		internalEnable			:= FALSE;		
		IF internalDisable THEN
			internalDisable		:= FALSE;
			internalState		:= MV_BEGIN_HALTING;
			
		// Reset all commands issued by method calls
		ELSIF fbMoveAbsCA[0].Busy OR fbMoveAbsCA[0].CommandAborted THEN // OR fbMoveAbs.CommandAborted THEN
			fbMoveAbsCA[0].Execute		:= FALSE;
		ELSIF fbMoveAbsCA[1].Busy OR fbMoveAbsCA[1].CommandAborted THEN
			fbMoveAbsCA[1].Execute		:= FALSE;			
		ELSIF fbAddToGroup.Done THEN
			fbAddToGroup.Execute		:= FALSE;
		ELSIF fbMoveRelCA[0].Busy OR fbMoveRelCA[0].CommandAborted THEN
			fbMoveRelCA[0].Execute		:= FALSE;
		ELSIF fbMoveRelCA[1].Busy OR fbMoveRelCA[1].CommandAborted THEN
			fbMoveRelCA[1].Execute		:= FALSE;
		ELSIF fbGearInPosMoverCA[0].Busy OR fbGearInPosMoverCA[0].CommandAborted THEN
			fbGearInPosMoverCA[0].Execute	:= FALSE;
		ELSIF fbGearInPosMoverCA[1].Busy OR fbGearInPosMoverCA[1].CommandAborted THEN
			fbGearInPosMoverCA[1].Execute	:= FALSE;
		ELSIF fbGearInPosAxisCA[0].Busy OR fbGearInPosAxisCA[0].CommandAborted THEN
			fbGearInPosAxisCA[0].Execute	:= FALSE;
		ELSIF fbGearInPosAxisCA[1].Busy OR fbGearInPosAxisCA[1].CommandAborted THEN
			fbGearInPosAxisCA[1].Execute	:= FALSE;
		ELSIF fbHaltCA.Busy OR fbHaltCA.CommandAborted OR fbHaltCA.Done THEN
			fbHaltCA.Execute			:= FALSE;
		// This is different than the other similar cases, since a Stop command should prevent other commands from overriding it, thus
		// the Execute needs to remain High until the command has fully completed.
		ELSIF fbGroupStop.Done THEN
			fbGroupStop.Execute			:= FALSE;
		END_IF;
		
		THIS^.CyclicTrack();
		
		IF (internalReissue) THEN
			THIS^.SourceInstancePath	:= 'ReissueCommand';

			CASE internalCurrentMoveType OF
				MOVETYPE_NONE:
					// No current command to reissue	
				MOVETYPE_POSITION:
					THIS^.MoveToPosition( internalCurrentDestPosition );
				MOVETYPE_STATION:
					THIS^.MoveToStation( internalCurrentDestStation );
				MOVETYPE_VELOCITY:
					THIS^.MoveVelocity( MotionParameters.Velocity );
				MOVETYPE_SYNC_MOVER:
					THIS^.SyncToMover( internalMasterMover, internalGap );
				MOVETYPE_SYNC_AXIS:
					// This command should perhaps not be compatible with Reissue command
			END_CASE
			internalReissue := FALSE;
		END_IF

		// And catch all internal function block errors
		IF fbMoveAbsCA[0].Error THEN
			ErrorID					:= fbMoveAbsCA[0].ErrorID;
			ErrorOrigin				:= CONCAT( InstancePath, '.fbMoveAbs[0]' );
			internalState			:= MV_ERROR;
		ELSIF fbMoveAbsCA[1].Error THEN
			ErrorID					:= fbMoveAbsCA[1].ErrorId;
			ErrorOrigin				:= CONCAT( InstancePath, '.fbMoveAbs[1]' );
			internalState			:= MV_ERROR;
		ELSIF fbAddToGroup.Error THEN
			ErrorID					:= fbAddToGroup.ErrorID;
			ErrorOrigin				:= CONCAT( InstancePath, '.fbAddToGroup' );
			internalState			:= MV_ERROR;
		ELSIF fbGroupStop.Error THEN
			ErrorID					:= fbGroupStop.ErrorId;
			ErrorOrigin				:= CONCAT( InstancePath, '.fbGroupStop' );
			internalState			:= MV_ERROR;
		ELSIF fbMoveRelCA[0].Error THEN
			ErrorID					:= fbMoveRelCA[0].ErrorID;
			ErrorOrigin 			:= CONCAT ( InstancePath, '.fbMoveRelCA[0]');
			internalState			:= MV_ERROR;
		ELSIF fbMoveRelCA[1].Error THEN
			ErrorID					:= fbMoveRelCA[1].ErrorID;
			ErrorOrigin 			:= CONCAT ( InstancePath, '.fbMoveRelCA[1]');
			internalState			:= MV_ERROR;
		ELSIF fbReadStatus.Valid AND fbReadStatus.ErrorStop THEN
			ErrorID					:= fbReadStatus.Status.ErrorID;
			ErrorOrigin				:= CONCAT( InstancePath, '.fbReadStatus' );
			internalState			:= MV_ERROR;
		ELSIF fbGearInPosMoverCA[0].Error THEN
			ErrorID					:= fbGearInPosMoverCA[0].ErrorId;
			ErrorOrigin				:= CONCAT( InstancePath, '.fbGearInPosMoverCA[0]');
			internalState			:= MV_ERROR;
		ELSIF fbGearInPosMoverCA[1].Error THEN
			ErrorID					:= fbGearInPosMoverCA[1].ErrorId;
			ErrorOrigin				:= CONCAT( InstancePath, '.fbGearInPosMoverCA[1]');
			internalState			:= MV_ERROR;
		ELSIF fbGearInPosAxisCA[0].Error THEN
			ErrorID					:= fbGearInPosAxisCA[0].ErrorId;
			ErrorOrigin				:= CONCAT( InstancePath, '.fbGearInPosAxisCA[0]');
			internalState			:= MV_ERROR;
		ELSIF fbGearInPosAxisCA[1].Error THEN
			ErrorID					:= fbGearInPosAxisCA[1].ErrorId;
			ErrorOrigin				:= CONCAT( InstancePath, '.fbGearInPosAxisCA[1]');
			internalState			:= MV_ERROR;			
		ELSIF fbActivateTrack.Error THEN
			ErrorID					:= fbActivateTrack.ErrorId;
			ErrorOrigin				:= CONCAT( InstancePath, '.fbActivateTrack');
			internalState			:= MV_ERROR;
		END_IF
		
	MV_BEGIN_HALTING:	// --------------------------------------------------- begin stopping process
	
		Ready	:= FALSE;
		Busy	:= TRUE;
		Error	:= FALSE;
		ErrorID	:= 0;
		
		// Kill any active motion commands
		fbMoveRelCA[0].Execute		:= FALSE;
		fbMoveRelCA[1].Execute		:= FALSE;
		fbMoveAbsCA[0].Execute		:= FALSE;
		fbMoveAbsCA[1].Execute		:= FALSE;
				
		IF fbReadStatus.ErrorStop = FALSE THEN
			fbHaltCA.Execute		:= TRUE;
			//fbHaltCA.Deceleration	:= MotionParameters.Deceleration;
			//fbHaltCA.Jerk			:= MotionParameters.Jerk;
		ELSE
			internalState			:= MV_REMOVEFROMGROUP;
		END_IF;
		
		IF fbHaltCA.Active OR fbHaltCA.Done THEN
			internalState			:= MV_HALTING;
		ELSIF fbHaltCA.Error THEN
			ErrorID					:= fbHaltCA.ErrorID;
			ErrorOrigin				:= CONCAT( InstancePath, '.fbHalt' );
			internalState			:= MV_ERROR;				
		END_IF	
		
	MV_HALTING:	// ------------------------------------------------------- mover disabling
	
		Ready	:= FALSE;
		Busy	:= TRUE;
		Error	:= FALSE;
		ErrorID	:= 0;

		// Wait for the stopping action to complete
		IF fbHaltCA.Done THEN
			fbHaltCA.Execute		:= FALSE;
			internalState			:= MV_REMOVEFROMGROUP;
		ELSIF fbHaltCA.Error THEN
			ErrorID					:= fbStop.ErrorID;
			ErrorOrigin				:= CONCAT( InstancePath, '.fbHalt' );
			internalState			:= MV_ERROR;
		END_IF	
		
	MV_REMOVEFROMGROUP:	// ---------------------------------------------------- remove mover from CA group
	
		Ready	:= FALSE;
		Busy	:= TRUE;
		Error	:= FALSE;
		ErrorID	:= 0;
		
		fbRemoveFromGroup.Execute			:= TRUE;
		fbRemoveFromGroup.IdentInGroup		:= UDINT_TO_IDENTINGROUP( IdentInGroup );
		
		IF fbRemoveFromGroup.Done THEN
			fbRemoveFromGroup.Execute		:= FALSE;
			internalState					:= MV_DISABLING;
		END_IF
		


	MV_DISABLING:	// ----------------------------------------------------- start the disabling process

		Ready	:= FALSE;
		Busy	:= TRUE;
		Error	:= FALSE;
		ErrorID	:= 0;
		
		fbPower.Enable				:= FALSE;
		fbPower.Enable_Positive		:= FALSE;
		fbPower.Enable_Negative		:= FALSE;
		fbPower.BufferMode			:= MC_Aborting;
		fbPower.Override			:= 100;
			
		IF fbPower.Status = FALSE THEN
			internalState			:= MV_IDLE;
		ELSIF fbPower.Error THEN
			ErrorID					:= fbPower.ErrorID;
			ErrorOrigin				:= CONCAT( InstancePath, '.fbPower' );
			internalState			:= MV_ERROR;
		END_IF		
	
	MV_ERROR: // ------------------------------------------------------- mover in error state
	
		Ready	:= FALSE;
		Busy	:= FALSE;
		Error	:= TRUE;
		
		internalEnable			:= FALSE;		
		IF internalDisable THEN
			internalDisable		:= FALSE;
			internalState		:= MV_REMOVEFROMGROUP;
			ErrorOrigin			:= '';
		END_IF
		
END_CASE

fbPower( Axis := AxisReference );
fbReset( Axis := AxisReference );
fbStop( Axis := AxisReference );

fbHaltCA( Axis := AxisReference );
//fbDisable( Axis := AxisRef );
//fbExternEnable( Axis := AxisRef );

fbAddToGroup( AxesGroup := GroupReference, Axis := AxisReference );
fbRemoveFromGroup( AxesGroup := GroupReference );

fbGroupStatus( AxesGroup := GroupReference );
fbGroupEnable( AxesGroup := GroupReference );
fbGroupReset( AxesGroup := GroupReference );
fbGroupStop( AxesGroup := GroupReference );

fbMoveAbsCA[0]( Axis := AxisReference );
fbMoveAbsCA[1]( Axis := AxisReference );
fbReadStatus( Enable := TRUE, Axis := AxisReference );
fbMoveRelCA[0] ( Axis := AxisReference );
fbMoveRelCA[1] ( Axis := AxisReference );

fbGearInPosMoverCA[0]( Master := internalMasterMover.AxisReference, Slave := THIS^.AxisReference );
fbGearInPosMoverCA[1]( Master := internalMasterMover.AxisReference, Slave := THIS^.AxisReference );

fbGearInPosAxisCA[0]( Master := internalMasterAxis, Slave := THIS^.AxisReference );
fbGearInPosAxisCA[1]( Master := internalMasterAxis, Slave := THIS^.AxisReference );

fbReadM1DetectMode();
fbReadM1DetectValid();
fbReadM1DetectActive();
fbWriteM1Detect();

// track management
fbActivateTrack(Axis := AxisReference);
fbReadTrackPositions(Axis := AxisReference);
END_METHOD

METHOD CyclicTrack : BOOL
VAR
END_VAR
VAR_INST
	MsgCreate			: FB_TcMessage;	
END_VAR
// called by .Cyclic() to handle the MC_ActivateTrack call's required state machine
// this is only called while the mover is in the RUN state within .Cyclic() by design
// calling the track management functions on disabled or errored movers that are not
// assigned to a group just causes the track management functions to throw more errors

CASE internalTrackState OF
	// wait for command
	TrackState.WAIT_FOR_COMMAND:
		IF (internalActivateTrackFlag) THEN
			// unregister mover from current track (logical tracking)
			IF (internalTrack <> 0) THEN
				internalTrack^.UnregisterMover(THIS^);
			END_IF;

			// set flags
			internalTrack := ADR(ErrorTrack);
			internalTrackIsReady := FALSE;

			// advance state
			internalTrackState := TrackState.SETUP_FUNCTION;
		END_IF
		
	// setup and call the function
	TrackState.SETUP_FUNCTION:
		fbActivateTrack.TrackId := internalActivatingTrack^.OTCID;
		fbActivateTrack.Execute := TRUE;
		IF (fbActivateTrack.Busy) THEN
			fbActivateTrack.Execute := FALSE;
			internalTrackState := TrackState.MONITOR_RESPONSE;
		END_IF
	
	// monitor response	
	TrackState.MONITOR_RESPONSE:
		IF (fbActivateTrack.Error) THEN
			internalTrackState := TrackState.ERROR;
		ELSIF (fbActivateTrack.Done) THEN
			internalTrackState := TrackState.REQUIRED_DELAY;
		END_IF;
	
	// required delay
	// the FB has returned .Done but the change has not yet propigated to the NC
	TrackState.REQUIRED_DELAY:
		internalTrackStateDelay.IN := TRUE;
		IF (internalTrackStateDelay.Q) THEN
			internalTrackStateDelay.IN := FALSE;
			internalTrackState := TrackState.CLEAN_UP;
		END_IF;
	
	// clean up flags
	TrackState.CLEAN_UP:
		internalTrack := internalActivatingTrack;
		internalActivatingTrack := ADR(ErrorTrack);
		internalTrackIsReady := TRUE;
		MsgCreate.CreateEx( TC_EVENTS.XtsBaseEventClass.MoverActivateTrackComplete, 0);
		MsgCreate.ipArguments.Clear().AddString(THIS^.InstancePath).AddInt(THIS^.CurrentTrack^.Id);
		MsgCreate.Send(0);
		internalTrackState := TrackState.WAIT_END;
		
	TrackState.ERROR:
		// reset execute
		fbActivateTrack.Execute := FALSE;
		// GVL.ERROR_TRACK is intentionally left in place
		// internalTrackIsReady is left at false
		// error is recorded in Cyclic()
		internalTrackState := TrackState.WAIT_END;
		
	TrackState.WAIT_END: 
		// falling edge detection for internalActivateTrackFlag
		IF (NOT internalActivateTrackFlag) THEN
			// register mover
			internalTrack^.RegisterMover(THIS^);
			internalTrackState := TrackState.WAIT_FOR_COMMAND;	
		END_IF
		internalActivateTrackFlag := FALSE;

END_CASE

// read back track information
IF (internalTrackIsReady) THEN
	// track info should be stable, call the block
	fbReadTrackPositions.Enable := TRUE;
	// copy data when ready
	IF (fbReadTrackPositions.Valid) THEN
		TrackInfo.TrackPosition := fbReadTrackPositions.TrackPosition;
		TrackInfo.PartPosition := fbReadTrackPositions.PartPosition;
		TrackInfo.TrackId := fbReadTrackPositions.TrackId;
		TrackInfo.PartId := fbReadTrackPositions.PartId;
	END_IF
ELSE
	// don't call function block to allow it to reset
	fbReadTrackPositions.Enable := FALSE;
END_IF


// a delay is required after MC_ActivateTrack returns .Done
internalTrackStateDelay(PT := T#10MS);
END_METHOD

METHOD Disable : iMover
VAR_INPUT
END_VAR
VAR
END_VAR
VAR_INST
	MsgCreate	: FB_TcMessage;	
END_VAR

IF internalState = MV_RUN OR internalState = MV_ERROR THEN

	// Sets an internal flag to advance the state machine
	internalDisable		:= TRUE;
	
	MsgCreate.CreateEx( TC_EVENTS.XtsBaseEventClass.MoverDisable,0 );
	MsgCreate.ipArguments.Clear().AddString(THIS^.InstancePath).AddString(THIS^.SourceInstancePath);
	MsgCreate.Send(0);	
END_IF

THIS^.SourceInstancePath	:= 'Direct access';

Disable		:= THIS^;
END_METHOD

METHOD Enable : iMover
VAR_INPUT
END_VAR
VAR
END_VAR
VAR_INST
	MsgCreate	: FB_TcMessage;	
END_VAR

IF internalState = MV_IDLE THEN

	// Sets an internal flag to advance the state machine
	internalEnable		:= TRUE;
	
	MsgCreate.CreateEx( TC_EVENTS.XtsBaseEventClass.MoverEnable,0 );
	MsgCreate.ipArguments.Clear().AddString(THIS^.InstancePath).AddString(THIS^.SourceInstancePath);
	MsgCreate.Send(0);

END_IF;

THIS^.SourceInstancePath	:= 'Direct access';

Enable := THIS^;
END_METHOD

METHOD GroupStop : iMover
VAR_INPUT
END_VAR
VAR
	newCallTime	: LREAL;
END_VAR
VAR_INST
	MsgCreate	: FB_TcMessage;	
END_VAR


IF NOT( Ready ) THEN	// if the mover is not ready & able to accept a GroupHalt Command

	internalState	:= MV_ERROR;
	ErrorID			:= 19201;

ELSE	// otherwise execute the command
	
	// grab a timestamp of the command
	newCallTime		:= ULINT_TO_LREAL(F_GetSystemTime())/1E7;
	
	fbGroupStop.Execute			:= TRUE;
	fbGroupStop.Deceleration	:= MotionParameters.Deceleration;
	fbGroupStop.Jerk			:= MotionParameters.Jerk;
	
	memset( ADR( internalCurrentDestObjective ), 0, SIZEOF( internalCurrentDestObjective ));
	internalCurrentMoveType		:= MoverCommandType_enum.MOVETYPE_NONE;
	
END_IF

IF ( newCallTime - lastCallGroupStop ) > 1 THEN
	MsgCreate.CreateEx( TC_EVENTS.XtsBaseEventClass.MoverGroupStop,0 );
	MsgCreate.ipArguments.Clear().AddString(THIS^.InstancePath).AddString(THIS^.SourceInstancePath);
	MsgCreate.Send(0);
END_IF

THIS^.SourceInstancePath	:= 'Direct access';

lastCallGroupStop	:= newCallTime;

GroupStop		:= THIS^;
END_METHOD

METHOD Halt : iMover
VAR_INPUT
END_VAR
VAR
	newCallTime: LREAL;
END_VAR
VAR_INST
	MsgCreate: FB_TcMessage;	
END_VAR

IF NOT( Ready ) THEN
	
	internalState	:= MV_ERROR;
	ErrorID			:= 19201;
	
ELSIF fbHaltCA.Busy THEN	

	newCallTime		:= ULINT_TO_LREAL(F_GetSystemTime())/1E7;
	
	// oddly, MC_HaltCA does not include an option for BufferMode
	// so do nothing
	
ELSE
	
	newCallTime		:= ULINT_TO_LREAL(F_GetSystemTime())/1E7;
	
	fbHaltCA.Execute		:= TRUE;
	fbHaltCA.Deceleration	:= MotionParameters.Deceleration;
	fbHaltCA.Jerk			:= MotionParameters.Jerk;
	
	fbHaltCA( Axis := AxisReference );
	
END_IF

internalCurrentMoveType		:= MOVETYPE_NONE;
internalCurrentDestPosition	:= 1E300;

memset( ADR( internalCurrentDestObjective), 0, SIZEOF( internalCurrentDestObjective ));
internalCurrentDestStation	REF= 0;

IF ( newCallTime - lastCallHalt ) > 1 THEN
	MsgCreate.CreateEx( TC_EVENTS.XtsBaseEventClass.MoverHalt,0);
	MsgCreate.ipArguments.Clear().AddString(THIS^.InstancePath).AddString(THIS^.SourceInstancePath).AddLReal(MotionParameters.Deceleration);
	MsgCreate.Send(0);
END_IF

THIS^.SourceInstancePath	:= 'Direct access';

lastCallHalt		:= newCallTIme;

Halt	:= THIS^;
END_METHOD

{attribute 'monitoring' := 'call'}
PROPERTY IsSyncedToAxis : BOOL
GET


IsSyncedToAxis		:= fbGearInPosAxisCA[0].InSync OR fbGearInPosAxisCA[1].InSync;
END_GET
END_PROPERTY

{attribute 'monitoring' := 'call'}
PROPERTY IsSyncedToMover : BOOL
GET


IsSyncedToMover		:= fbGearInPosMoverCA[0].InSync OR fbGearInPosMoverCA[1].InSync;
END_GET
END_PROPERTY

PROPERTY IsTrackReady : BOOL
GET
IsTrackReady := internalTrackIsReady;
END_GET
END_PROPERTY

METHOD LogUserEvent : iMover
VAR_INPUT
	String1	: STRING;	// First content section of user-event message
	String2 : STRING;	// Second content section of user-event message
	String3 : STRING;	// Third content section of user-event message
END_VAR
VAR
END_VAR
VAR_INST
	MsgCreate: FB_TcMessage;	
END_VAR



MsgCreate.CreateEx( TC_EVENTS.XtsBaseEventClass.UserEvent, 0 );
MsgCreate.ipArguments.Clear().AddString(String1).AddString(String2).AddString(String3);
MsgCreate.Send(0);

LogUserEvent	:= THIS^;
END_METHOD

PROPERTY MasterMover : Reference To Mover
GET


IF THIS^.internalCurrentMoveType = MOVETYPE_SYNC_MOVER THEN
	MasterMover		REF= internalMasterMover;
ELSE
	MasterMover		REF= 0;
END_IF
END_GET
END_PROPERTY

METHOD PUBLIC MoveToPosition : iMover
VAR_INPUT
	DestinationPosition		: LREAL;	// position on track for a shuttle to move towards
END_VAR
VAR
	newCallTime		: LREAL;
END_VAR
VAR_INST
	MsgCreate		: FB_TcMessage;	
END_VAR

IF NOT( Ready ) THEN	// if the mover is not ready & able to accept a moveabs command...
	
	internalState	:= MV_ERROR;
	ErrorID			:= 19201;
	
ELSE	// otherwise let 'er rip
	
	newCallTime		:= ULINT_TO_LREAL(F_GetSystemTime())/1E7;
	internalReissue := FALSE;	// reissue no longer necessary
	
	IF fbMoveAbsCA[0].Busy = FALSE THEN
		
		fbMoveAbsCA[0].Jerk			:= MotionParameters.Jerk;
		fbMoveAbsCA[0].Acceleration	:= MotionParameters.Acceleration;
		fbMoveAbsCA[0].Deceleration	:= MotionParameters.Deceleration;
		fbMoveAbsCA[0].Velocity		:= MotionParameters.Velocity;
		fbMoveAbsCA[0].Direction	:= MotionParameters.Direction;
		fbMoveAbsCA[0].Options.DynamicsReferenceSystem := CurrentTrack^.OTCID;
		fbMoveAbsCA[0].Options.PositionReferenceSystem := CurrentTrack^.OTCID;
		
		fbMoveAbsCA[0].Position		:= DestinationPosition;
		
		fbMoveAbsCA[0].BufferMode	:= mcAborting;
		fbMoveAbsCA[0].Execute		:= TRUE;
		 
		fbMoveAbsCA[0].Execute		:= TRUE;		// execute this block, and...
		fbMoveAbsCA[1].Execute		:= FALSE;		// if necessary, interrupt this one
		
		fbMoveAbsCA[0]( Axis := AxisReference );
		
	ELSIF fbMoveAbsCA[1].Busy = FALSE THEN
		
		fbMoveAbsCA[1].Jerk			:= MotionParameters.Jerk;
		fbMoveAbsCA[1].Acceleration	:= MotionParameters.Acceleration;
		fbMoveAbsCA[1].Deceleration	:= MotionParameters.Deceleration;
		fbMoveAbsCA[1].Velocity		:= MotionParameters.Velocity;
		fbMoveAbsCA[1].Direction	:= MotionParameters.Direction;
		fbMoveAbsCA[1].Options.DynamicsReferenceSystem := CurrentTrack^.OTCID;
		fbMoveAbsCA[1].Options.PositionReferenceSystem := CurrentTrack^.OTCID;

		
		fbMoveAbsCA[1].Position		:= DestinationPosition;
		
		fbMoveAbsCA[1].BufferMode	:= mcAborting;
		fbMoveAbsCA[1].Execute		:= TRUE;
		
		fbMoveAbsCA[1].Execute		:= TRUE;		// execute this block, and...
		fbMoveAbsCA[0].Execute		:= FALSE;		// if necessary, interrupt this one
		
		fbMoveAbsCA[1]( Axis := AxisReference );
		 
	ELSE
		MsgCreate.CreateEx( TC_EVENTS.XtsBaseEventClass.MoverMoveToPositionOverload,0 );
		MsgCreate.ipArguments.Clear().AddString(THIS^.InstancePath).AddString(THIS^.SourceInstancePath).AddLReal(DestinationPosition);
		MsgCreate.Send(0);
	END_IF
	
END_IF

internalCurrentMoveType		:= MOVETYPE_POSITION;
internalCurrentDestPosition := DestinationPosition;

memset( ADR( internalCurrentDestObjective ), 0, SIZEOF( internalCurrentDestObjective ));
internalCurrentDestStation	REF= 0;

IF ( newCallTime - lastCallMovePos ) > 1 THEN
	MsgCreate.CreateEx( TC_EVENTS.XtsBaseEventClass.MoverMoveToPosition,0 );
	MsgCreate.ipArguments.Clear().AddString(THIS^.InstancePath).AddString(THIS^.SourceInstancePath).AddLReal(DestinationPosition);
	MsgCreate.Send(0);
END_IF;

THIS^.SourceInstancePath	:= 'Direct access';

lastCallMovePos		:= newCallTime;

MoveToPosition		:= THIS^;
END_METHOD

METHOD MoveToStation : iMover
VAR_INPUT
	DestinationStation	: REFERENCE TO Station;	
END_VAR
VAR
	newCallTime			: LREAL;
END_VAR
VAR_INST
	MsgCreate			: FB_TcMessage;	
END_VAR
IF NOT( Ready ) AND NOT(__ISVALIDREF( DestinationStation )) THEN	// if the mover is not ready & able to accept a moveabs command...
	
	internalState	:= MV_ERROR;
	ErrorID			:= 19201;
	
ELSE	// otherwise let 'er rip
	
	newCallTime		:= ULINT_TO_LREAL(F_GetSystemTime())/1E7;
	internalReissue := FALSE;	// reissue no longer necessary
	
	IF fbMoveAbsCA[0].Busy = FALSE THEN
		
		fbMoveAbsCA[0].Jerk			:= MotionParameters.Jerk;
		fbMoveAbsCA[0].Acceleration	:= MotionParameters.Acceleration;
		fbMoveAbsCA[0].Deceleration	:= MotionParameters.Deceleration;
		fbMoveAbsCA[0].Velocity		:= MotionParameters.Velocity;
		fbMoveAbsCA[0].Direction	:= MotionParameters.Direction;
		fbMoveAbsCA[0].Options.DynamicsReferenceSystem := CurrentTrack^.OTCID;
		fbMoveAbsCA[0].Options.PositionReferenceSystem := CurrentTrack^.OTCID;
		
		fbMoveAbsCA[0].Position		:= DestinationStation.internalPosition;
		
		fbMoveAbsCA[0].BufferMode	:= mcAborting;
		fbMoveAbsCA[0].Execute		:= TRUE;
		 
		fbMoveAbsCA[0].Execute		:= TRUE;		// execute this block, and...
		fbMoveAbsCA[1].Execute		:= FALSE;		// if necessary, interrupt this one
		
		fbMoveAbsCA[0]( Axis := AxisReference );
		
	ELSIF fbMoveAbsCA[1].Busy = FALSE THEN
		
		fbMoveAbsCA[1].Jerk			:= MotionParameters.Jerk;
		fbMoveAbsCA[1].Acceleration	:= MotionParameters.Acceleration;
		fbMoveAbsCA[1].Deceleration	:= MotionParameters.Deceleration;
		fbMoveAbsCA[1].Velocity		:= MotionParameters.Velocity;
		fbMoveAbsCA[1].Direction	:= MotionParameters.Direction;
		fbMoveAbsCA[1].Options.DynamicsReferenceSystem := CurrentTrack^.OTCID;
		fbMoveAbsCA[1].Options.PositionReferenceSystem := CurrentTrack^.OTCID;
		
		fbMoveAbsCA[1].Position		:= DestinationStation.internalPosition;
		
		fbMoveAbsCA[1].BufferMode	:= mcAborting;
		fbMoveAbsCA[1].Execute		:= TRUE;
		
		fbMoveAbsCA[1].Execute		:= TRUE;		// execute this block, and...
		fbMoveAbsCA[0].Execute		:= FALSE;		// if necessary, interrupt this one

		fbMoveAbsCA[1]( Axis := AxisReference );	

	ELSE
		MsgCreate.CreateEx( TC_EVENTS.XtsBaseEventClass.MoverMoveToStationOverload,0 );
		MsgCreate.ipArguments.Clear().AddString(THIS^.InstancePath).AddString(THIS^.SourceInstancePath).AddString(DestinationStation.InstancePath);
		MsgCreate.Send(0);
		
	END_IF
	
	// Set the current destination object to the instance path of the objective, or 0 if unassigned
	internalCurrentDestPosition		:= DestinationStation.Position;
	internalCurrentDestObjective	:= SEL( __ISVALIDREF( DestinationStation ), '', DestinationStation.InstancePath );
	internalCurrentDestStation		REF= DestinationStation;
	internalCurrentMoveType			:= MOVETYPE_STATION;
	
	// Register this mover with the station, so the station knows this mover is incoming
	DestinationStation.RegisterMover( THIS^ );
	
END_IF

IF ( newCallTime - lastCallMoveSta ) > 1 THEN
	MsgCreate.CreateEx( TC_EVENTS.XtsBaseEventClass.MoverMoveToStation,0 );
	MsgCreate.ipArguments.Clear().AddString(THIS^.InstancePath).AddString(THIS^.SourceInstancePath).AddString(DestinationStation.InstancePath);
	MsgCreate.Send(0);
END_IF

THIS^.SourceInstancePath	:= 'Direct access';

lastCallMoveSta		:= newCallTime;

MoveToStation		:= THIS^;
END_METHOD

METHOD MoveVelocity : iMover
VAR_INPUT
	DesiredVelocity : LREAL;		//The velocity to be commanded [mm/s]
END_VAR
VAR
	negativeCommand	: BOOL;
	newCallTime		: LREAL;
END_VAR
VAR_INST
	MsgCreate		: FB_TcMessage;	
END_VAR
IF NOT ( ready ) THEN
	
	internalState	:= MV_ERROR;
	ErrorID			:= 19201;
	
ELSE
	
	newCallTime		:= ULINT_TO_LREAL(F_GetSystemTime())/1E7;
	internalReissue := FALSE;	// reissue no longer necessary
	
	negativeCommand					:= SEL( DesiredVelocity < 0, FALSE, TRUE );
	MotionParameters.Velocity		:= ABS( DesiredVelocity );
	
	IF fbMoveRelCA[0].Busy = FALSE THEN
		
		fbMoveRelCA[0].Jerk			:= MotionParameters.Jerk;
		
		fbMoveRelCA[0].Acceleration	:= MotionParameters.Acceleration;
		fbMoveRelCA[0].Deceleration	:= MotionParameters.Deceleration;
		fbMoveRelCA[0].Velocity		:= MotionParameters.Velocity;
		
		fbMoveRelCA[0].Distance		:= SEL( negativeCommand, 1E100, -1E100 );
		
		      
		fbMoveRelCA[0].BufferMode	:= mcAborting;
		      
		fbMoveRelCA[0].Execute		:= TRUE;		// execute this block, and...
		fbMoveRelCA[1].Execute		:= FALSE;		// if necessary, interrupt this one
		
		fbMoveRelCA[0]( Axis := AxisReference );
		
	ELSIF fbMoveRelCA[1].Busy = FALSE THEN
		
		fbMoveRelCA[1].Jerk			:= MotionParameters.Jerk;
		
		fbMoveRelCA[1].Acceleration	:= MotionParameters.Acceleration;
		fbMoveRelCA[1].Deceleration	:= MotionParameters.Deceleration;
		fbMoveRelCA[1].Velocity		:= MotionParameters.Velocity;
		      
		fbMoveRelCA[1].Distance		:= SEL( negativeCommand, 1E100, -1E100 );
		      
		fbMoveRelCA[1].BufferMode	:= mcAborting;
		      
		fbMoveRelCA[1].Execute		:= TRUE;		// execute this block, and...
		fbMoveRelCA[0].Execute		:= FALSE;		// if necessary, interrupt this one

		fbMoveRelCA[1]( Axis := AxisReference );
	ELSE
		MsgCreate.CreateEx( TC_EVENTS.XtsBaseEventClass.MoverMoveVelocityOverload,0 );
		MsgCreate.ipArguments.Clear().AddString(THIS^.InstancePath).AddString(THIS^.SourceInstancePath).AddLReal(DesiredVelocity);
		MsgCreate.Send(0);
	END_IF

END_IF

fbMoveRelCA[0] ( Axis := AxisReference );
fbMoveRelCA[1] ( Axis := AxisReference );


internalCurrentMoveType		:= MOVETYPE_VELOCITY;
internalCurrentDestPosition := 1E300;

memset( ADR( internalCurrentDestObjective ), 0, SIZEOF( internalCurrentDestObjective ));
internalCurrentDestStation	REF= 0;

IF ( newCallTime - lastCallMoveVel ) > 1 THEN
	MsgCreate.CreateEx( TC_EVENTS.XtsBaseEventClass.MoverMoveVelocity,0 );
	MsgCreate.ipArguments.Clear().AddString(THIS^.InstancePath).AddString(THIS^.SourceInstancePath).AddLReal(DesiredVelocity);
	MsgCreate.Send(0);
END_IF;

THIS^.SourceInstancePath	:= 'Direct access';

lastCallMoveVel		:= newCallTime;

MoveVelocity		:= THIS^;
END_METHOD

PROPERTY Payload : Payload_TYP;
GET


Payload	:= internalPayload;
END_GET
SET


internalPayload	:= Payload;
END_SET
END_PROPERTY

METHOD ReissueCommand : iMover
VAR_INPUT
END_VAR

// set flag for use in .Cyclic()
internalReissue := TRUE;


ReissueCommand		:= THIS^;
END_METHOD

METHOD SetAcceleration : iMover
VAR_INPUT
	Acceleration	: LREAL;
END_VAR
VAR
	newCallTime		: LREAL;
END_VAR
VAR_INST
	MsgCreate		: FB_TcMessage;	
END_VAR

newCallTime		:= ULINT_TO_LREAL(F_GetSystemTime())/1E7;

MotionParameters.Acceleration		:= LIMIT( 0, Acceleration, 1E300 );	// upper limit is capped by the axis object parameters

THIS^.ReissueCommand();

IF ( newCallTime - lastCallSetAcc ) > 1 THEN
	MsgCreate.CreateEx( TC_EVENTS.XtsBaseEventClass.MoverSetAcceleration,0 );
	MsgCreate.ipArguments.Clear().AddString(THIS^.InstancePath).AddString(THIS^.SourceInstancePath).AddLReal(Acceleration);
	MsgCreate.Send(0);
END_IF;

THIS^.SourceInstancePath	:= 'Direct access';

lastCallSetAcc		:= newCallTime;

SetAcceleration		:= THIS^;
END_METHOD

METHOD SetDeceleration : iMover
VAR_INPUT
	Deceleration	: LREAL;
END_VAR
VAR
	newCallTime		: LREAL;
END_VAR
VAR_INST
	MsgCreate		: FB_TcMessage;	
END_VAR

newCallTime		:= ULINT_TO_LREAL(F_GetSystemTime())/1E7;

MotionParameters.Deceleration	:= LIMIT( 0, Deceleration, 1E300 ); // upper limit is capped by the axis parameters

THIS^.ReissueCommand();

IF ( newCallTime - lastCallSetDec ) > 1 THEN
	MsgCreate.CreateEx( TC_EVENTS.XtsBaseEventClass.MoverSetDeceleration,0 );
	MsgCreate.ipArguments.Clear().AddString(THIS^.InstancePath).AddString(THIS^.SourceInstancePath).AddLReal(Deceleration);
	MsgCreate.Send(0);
END_IF

THIS^.SourceInstancePath	:= 'Direct access';

lastCallSetDec		:= newCallTime;

SetDeceleration		:= THIS^;
END_METHOD

METHOD SetDirection : iMover
VAR_INPUT
	Direction		: Tc3_Mc3Definitions.MC_Direction;
END_VAR
VAR
	newCallTime		: LREAL;
END_VAR
VAR_INST
	MsgCreate		: FB_TcMessage;	
END_VAR

newCallTime		:= ULINT_TO_LREAL(F_GetSystemTime())/1E7;

MotionParameters.Direction		:= Direction;

THIS^.ReissueCommand();

IF ( newCallTime - lastCallSetDir ) > 1 THEN
	MsgCreate.CreateEx( TC_EVENTS.XtsBaseEventClass.MoverSetDirection,0 );
	MsgCreate.ipArguments.Clear().AddString(THIS^.InstancePath).AddString(THIS^.SourceInstancePath).AddInt(Direction);
	MsgCreate.Send(0);
END_IF

THIS^.SourceInstancePath	:= 'Direct access';

lastCallSetDir		:= newCallTime;

SetDirection		:= THIS^;
END_METHOD

METHOD SetJerk : iMover
VAR_INPUT
	Jerk		: LREAL;
END_VAR
VAR
	newCallTime	: LREAL;
END_VAR
VAR_INST
	MsgCreate	: FB_TcMessage;	
END_VAR

newCallTime		:= ULINT_TO_LREAL(F_GetSystemTime())/1E7;

MotionParameters.Jerk		:= LIMIT( 0, Jerk, 1E300 ); // upper limit is capped by the axis parameters

THIS^.ReissueCommand();

IF ( newCallTime - lastCallSetJerk ) > 1 THEN
	MsgCreate.CreateEx( TC_EVENTS.XtsBaseEventClass.MoverSetJerk,0 );
	MsgCreate.ipArguments.Clear().AddString(THIS^.InstancePath).AddString(THIS^.SourceInstancePath).AddLReal(Jerk);
	MsgCreate.Send(0);
END_IF

THIS^.SourceInstancePath	:= 'Direct access';

lastCallSetJerk		:= newCallTIme;

SetJerk		:= THIS^;
END_METHOD

METHOD SetVelocity : iMover
VAR_INPUT
	Velocity		: LREAL;		// Updates Mover's internal velocity parameter. Takes effect immediately. [mm/s]
END_VAR
VAR
	logstr			: STRING(200);		// method variable containing an event log message for the command
	LogEvent		: INT;
	newCallTime		: LREAL;
END_VAR
VAR_INST
	MsgCreate		: FB_TcMessage;	
END_VAR

newCallTime		:= ULINT_TO_LREAL(F_GetSystemTime())/1E7;

MotionParameters.Velocity	:= LIMIT( 0, Velocity, 1E300 ); // upper limit is capped by the axis parameters 

THIS^.ReissueCommand();

IF ( newCallTime - lastCallSetVel ) > 1 THEN
	MsgCreate.CreateEx( TC_EVENTS.XtsBaseEventClass.MoverSetVelocity,0 );
	MsgCreate.ipArguments.Clear().AddString(THIS^.InstancePath).AddString(THIS^.SourceInstancePath).AddLReal(Velocity);
	MsgCreate.Send(0);
END_IF

THIS^.SourceInstancePath	:= 'Direct access';

lastCallSetVel	:= newCallTime;

SetVelocity		:= THIS^;
END_METHOD

METHOD SyncToAxis : iMover
VAR_INPUT
	
	MasterAxis		: REFERENCE TO AXIS_REF;
	MasterSyncPos	: LREAL;				// Master sync position (nonmodulo), where the input axis will be located when first synchronized
	SlaveSyncPos	: LREAL;				// Mover sync position, where the mover will be located when first synchronized
	SyncStrategy	: MC_SYNC_STRATEGY;		// Direction input
	
END_VAR
VAR
	newCallTime		: LREAL;
END_VAR
VAR_INST
	MsgCreate		: FB_TcMessage;
END_VAR


IF NOT( Ready ) THEN
	
	internalState		:= MV_ERROR;
	ErrorID				:= 19201;
	
ELSE
	
	newCallTime			:= ULINT_TO_LREAL(F_GetSystemTime())/1E7;
	internalReissue := FALSE;	// reissue no longer necessary
	
	internalMasterAxis		REF= MasterAxis;
	
	IF fbGearInPosAxisCA[0].Busy = FALSE THEN
		
		fbGearInPosAxisCA[0].Execute			:= TRUE;
		
		fbGearInPosAxisCA[0].RatioNumerator		:= 1;
		fbGearInPosAxisCA[0].RatioDenumerator	:= 1;
		
		fbGearInPosAxisCA[0].MasterSyncPosition	:= MasterSyncPos;	// This needs to be nonmodulo
		fbGearInPosAxisCA[0].SlaveSyncPosition	:= SlaveSyncPos;
		
		fbGearInPosAxisCA[0].SyncStrategy		:= SyncStrategy;
		
		fbGearInPosAxisCA[0].Options.DynamicsReferenceSystem := CurrentTrack^.OTCID;
		fbGearInPosAxisCA[0].Options.SlaveSyncPositionReferenceSystem := CurrentTrack^.OTCID;

		
		IF MotionParameters.Direction = mcDirectionPositive THEN
			fbGearInPosAxisCA[0].SyncMode		:= mcSyncModePositive;
		ELSIF MotionParameters.Direction = mcDirectionNegative THEN
			fbGearInPosAxisCA[0].SyncMode		:= mcSyncModeNegative;
		END_IF
		
		fbGearInPosAxisCA[0].Velocity			:= MotionParameters.Velocity;
		fbGearInPosAxisCA[0].Acceleration		:= MotionParameters.Acceleration;
		fbGearInPosAxisCA[0].Deceleration		:= MotionParameters.Deceleration;
		fbGearInPosAxisCA[0].Jerk				:= MotionParameters.Jerk;
		
		fbGearInPosAxisCA[0].BufferMode			:= Tc3_Mc3Definitions.MC_BUFFER_MODE.mcAborting;
		
		fbGearInPosAxisCA[0]( Master := MasterAxis, Slave := THIS^.AxisReference );		
		
	ELSIF fbGearInPosAxisCA[1].Busy = FALSE THEN
		
		fbGearInPosAxisCA[1].Execute			:= TRUE;
		
		fbGearInPosAxisCA[1].RatioNumerator		:= 1;
		fbGearInPosAxisCA[1].RatioDenumerator	:= 1;
		
		fbGearInPosAxisCA[1].MasterSyncPosition	:= MasterSyncPos;	// This needs to be nonmodulo
		fbGearInPosAxisCA[1].SlaveSyncPosition	:= SlaveSyncPos;
		
		fbGearInPosAxisCA[1].SyncStrategy		:= SyncStrategy;
		
		fbGearInPosAxisCA[1].Options.DynamicsReferenceSystem := CurrentTrack^.OTCID;
		fbGearInPosAxisCA[1].Options.SlaveSyncPositionReferenceSystem := CurrentTrack^.OTCID;
		
		IF MotionParameters.Direction = mcDirectionPositive THEN
			fbGearInPosAxisCA[1].SyncMode		:= mcSyncModePositive;
		ELSIF MotionParameters.Direction = mcDirectionNegative THEN
			fbGearInPosAxisCA[1].SyncMode		:= mcSyncModeNegative;				
		END_IF
		
		fbGearInPosAxisCA[1].Velocity			:= MotionParameters.Velocity;
		fbGearInPosAxisCA[1].Acceleration		:= MotionParameters.Acceleration;
		fbGearInPosAxisCA[1].Deceleration		:= MotionParameters.Deceleration;
		fbGearInPosAxisCA[1].Jerk				:= MotionParameters.Jerk;
		
		fbGearInPosAxisCA[1].BufferMode			:= Tc3_Mc3Definitions.MC_BUFFER_MODE.mcAborting;
		
		fbGearInPosAxisCA[1]( Master := MasterAxis, Slave := THIS^.AxisReference );

	ELSE
		MsgCreate.CreateEx( TC_EVENTS.XtsBaseEventClass.MoverSyncToAxisOverload, 0 );
		MsgCreate.ipArguments.Clear().AddString(THIS^.InstancePath).AddString(THIS^.SourceInstancePath);
		MsgCreate.Send(0);
	END_IF
	
END_IF

internalCurrentMoveType			:= MOVETYPE_SYNC_AXIS;
internalCurrentDestPosition		:= 1E300;

memset( ADR( internalCurrentDestObjective ), 0, SIZEOF( internalCurrentDestObjective ));
internalCurrentDestStation		REF= 0;

IF ( newCallTime - lastCallSync ) > 1 THEN
	MsgCreate.CreateEx( TC_EVENTS.XtsBaseEventClass.MoverSyncToAxis, 0 );
	MsgCreate.ipArguments.Clear().AddString(THIS^.InstancePath).AddString(THIS^.SourceInstancePath);
	MsgCreate.Send(0);
END_IF

THIS^.SourceInstancePath		:= 'Direct access';

lastCallSync	:= newCallTime;

SyncToAxis		:= THIS^;
END_METHOD

METHOD SyncToMover : iMover
VAR_INPUT
	MasterMover			: REFERENCE TO Mover;	// Synchronization master mover, whose position to follow. Further motion commands break the pairing
	Gap					: LREAL;				// Gap distance to lead mover. Positive values indicate following, negative values indicate leading
END_VAR
VAR
	CWDistToSync		: LREAL;
	CWDistToMaster		: LREAL;
	syncPos				: LREAL;
	newCallTime			: LREAL;
END_VAR
VAR_INST
	MsgCreate			: FB_TcMessage;	
END_VAR
IF NOT( Ready ) THEN

	internalState	:= MV_ERROR;
	ErrorID			:= 19201;
	
ELSE	// let 'er rip
	
	newCallTime		:= ULINT_TO_LREAL(F_GetSystemTime())/1E7;
	internalReissue := FALSE;	// reissue no longer necessary

	internalMasterMover		REF= MasterMover;
	internalGap				:= Gap;
	
	
	syncPos			:= internalMasterMover.AxisReference.NcToPlc.ActPos - internalGap;
	CWDistToSync	:= MODABS( syncPos - THIS^.AxisReference.NcToPlc.ActPos, GVL.TRACK_LENGTH );
	CWDistToMaster	:= MODABS( internalMasterMover.AxisReference.NcToPlc.ActPos - THIS^.AxisReference.NcToPlc.ActPos, GVL.TRACK_LENGTH );
		
	IF fbGearInPosMoverCA[0].Busy = FALSE THEN
		
		fbGearInPosMoverCA[0].Execute				:= TRUE;
			
		fbGearInPosMoverCA[0].RatioNumerator			:= 1;
		fbGearInPosMoverCA[0].RatioDenumerator		:= 1;
		
		fbGearInPosMoverCA[0].MasterSyncPosition		:= internalMasterMover.AxisReference.NcToPlc.ActPos;
		fbGearInPosMoverCA[0].SlaveSyncPosition		:= MODABS( internalMasterMover.AxisReference.NcToPlc.ActPos - internalGap, GVL.TRACK_LENGTH);
		
		fbGearInPosMoverCA[0].SyncStrategy			:= mcSyncStrategyEarly;		
		fbGearInPosMoverCA[0].SyncMode				:= SEL( CWDistToSync < CWDistToMaster, mcSyncModeNegative, mcSyncModePositive );
				
		//fbGearInPosMoverCA[0].Options.MinimalSlavePosition	:= -1E300;
		
		fbGearInPosMoverCA[0].Velocity				:= MotionParameters.Velocity;
		fbGearInPosMoverCA[0].Acceleration			:= MotionParameters.Acceleration;
		fbGearInPosMoverCA[0].Deceleration			:= MotionParameters.Deceleration;
		fbGearInPosMoverCA[0].Jerk					:= MotionParameters.Jerk;
		
		fbGearInPosMoverCA[0].BufferMode				:= Tc3_Mc3Definitions.MC_BUFFER_MODE.mcAborting;
		
		fbGearInPosMoverCA[0]( Master := internalMasterMover.AxisReference, Slave := THIS^.AxisReference );
		
	ELSIF fbGearInPosMoverCA[1].Busy = FALSE THEN
		
		fbGearInPosMoverCA[1].Execute				:= TRUE;
		
		fbGearInPosMoverCA[1].RatioNumerator			:= 1;
		fbGearInPosMoverCA[1].RatioDenumerator		:= 1;
		
		fbGearInPosMoverCA[1].MasterSyncPosition		:= internalMasterMover.AxisReference.NcToPlc.ActPos;
		fbGearInPosMoverCA[1].SlaveSyncPosition		:= MODABS( internalMasterMover.AxisReference.NcToPlc.ActPos - internalGap, GVL.TRACK_LENGTH);
		
		fbGearInPosMoverCA[1].SyncStrategy			:= mcSyncStrategyEarly;
		fbGearInPosMoverCA[1].SyncMode				:= SEL( CWDistToSync < CWDistToMaster, mcSyncModeNegative, mcSyncModePositive );
		
		//fbGearInPosMoverCA[1].Options.MinimalSlavePosition	:= -1E300;
		
		fbGearInPosMoverCA[1].Velocity				:= MotionParameters.Velocity;
		fbGearInPosMoverCA[1].Acceleration			:= MotionParameters.Acceleration;
		fbGearInPosMoverCA[1].Deceleration			:= MotionParameters.Deceleration;
		fbGearInPosMoverCA[1].Jerk					:= MotionParameters.Jerk;
		
		fbGearInPosMoverCA[1].BufferMode				:= Tc3_Mc3Definitions.MC_BUFFER_MODE.mcAborting;
		
		
		fbGearInPosMoverCA[1]( Master := internalMasterMover.AxisReference, Slave := THIS^.AxisReference );
		
	ELSE
		MsgCreate.CreateEx( TC_EVENTS.XtsBaseEventClass.MoverSyncToMoverOverload,0 );
		MsgCreate.ipArguments.Clear().AddString(THIS^.InstancePath).AddString(THIS^.SourceInstancePath).AddString(MasterMover.InstancePath).AddLReal(Gap);
		MsgCreate.Send(0);
		
	END_IF

END_IF;

internalCurrentMoveType			:= MOVETYPE_SYNC_MOVER;
internalCurrentDestPosition		:= 1E300;

memset( ADR( internalCurrentDestObjective ), 0, SIZEOF( internalCurrentDestObjective ));
internalCurrentDestStation	REF= 0;

IF ( newCallTime - lastCallSync ) > 1 THEN
	MsgCreate.CreateEx( TC_EVENTS.XtsBaseEventClass.MoverSyncToMover,0 );
	MsgCreate.ipArguments.Clear().AddString(THIS^.InstancePath).AddString(THIS^.SourceInstancePath).AddString(MasterMover.InstancePath).AddLReal(Gap);
	MsgCreate.Send(0);
END_IF

THIS^.SourceInstancePath	:= 'Direct access';

lastCallSync		:= newCallTime;


SyncToMover		:= THIS^;
END_METHOD

END_FUNCTION_BLOCK

// ---- POUs/XTS/Station.TcPOU
FUNCTION_BLOCK Station EXTENDS Objective
VAR

    {attribute 'hide'}
    internalPosition : LREAL;
	internalTrackId : DINT := 1; 

END_VAR

{attribute 'monitoring' := 'variable'}
PROPERTY CurrentMover : REFERENCE TO Mover
GET
VAR

    i          : ULINT;
    difference : LREAL;

	moverTrackId: INT;
END_VAR
// default to unassigned
CurrentMover REF= 0;

FOR i := 0 TO SIZEOF(internalTrackedMovers) / SIZEOF(internalTrackedMovers[0]) - 1 DO

    // In order to deal with the rollover, we need to evaluate distance between congruence classes
    // e.g. On a 4m track, if the Station is at 0.34mm and the Mover is at 3999.8mm, then this is considered 'in position'	

    IF internalTrackedMovers[i] <> 0 THEN
		moverTrackId := internalTrackedMovers[i]^.CurrentTrack^.Id;
		IF (moverTrackId = internalTrackId) THEN

			difference := ABS(internalTrackedMovers[i]^.TrackInfo.TrackPosition - Position);

			IF MIN(difference, GVL.TRACK_LENGTH - difference) < 1.0 AND NOT internalTrackedMovers[i]^.Busy THEN
				CurrentMover                    REF= internalTrackedMovers[i]^;
				CurrentMover.SourceInstancePath := THIS^.InstancePath;
			END_IF
		END_IF
    END_IF

END_FOR

// If the Station has no CurrentMover, then return an imposter ErrorMover, whose method calls all trigger an error message
IF __ISVALIDREF(CurrentMover) = FALSE THEN
    ErrorMover.SourceInstancePath := THIS^.InstancePath;
    CurrentMover                  REF= ErrorMover;
END_IF
END_GET
END_PROPERTY

METHOD Cyclic : BOOL

VAR
    i : USINT;
END_VAR
FOR i := 0 TO GVL.NUM_MOVERS - 1 DO

    // This mover is no longer destined for any station
    IF internalTrackedMovers[i] <> 0 AND_THEN internalTrackedMovers[i]^.CurrentMoveType <> MOVETYPE_STATION THEN
        internalTrackedMovers[i] := 0;
        // This mover is no longer destined for this specific station. Comparing instance path seems to be the best way to do this comparison?
    ELSIF internalTrackedMovers[i] <> 0 AND_THEN internalTrackedMovers[i]^.CurrentObjective <> InstancePath THEN
        internalTrackedMovers[i] := 0;
    END_IF

END_FOR
END_METHOD

{attribute 'monitoring' := 'variable'}
PROPERTY MoverInPosition : BOOL
GET
VAR

    i          : ULINT;
    difference : LREAL;
	moverTrackId: INT;
END_VAR
// default to false
MoverInPosition := FALSE;

FOR i := 0 TO SIZEOF(internalTrackedMovers) / SIZEOF(internalTrackedMovers[0]) - 1 DO

    // In order to deal with the rollover, we need to evaluate distance between congruence classes
    // e.g. On a 4m track, if the Station is at 0.34 mm and the Mover is at 3999.8mm, then this is considered 'in position' 

    // todo: make in-position tolerance adjustable. add condition that mover is stopped?
    IF internalTrackedMovers[i] <> 0 THEN
		moverTrackId := internalTrackedMovers[i]^.CurrentTrack^.Id;
		IF (moverTrackId = internalTrackId) THEN
			difference := Position - internalTrackedMovers[i]^.TrackInfo.TrackPosition;

			IF MIN(difference, GVL.TRACK_LENGTH - difference) < 1.0 AND NOT internalTrackedMovers[i]^.Busy THEN
				MoverInPosition := TRUE;
			END_IF
		END_IF;
    END_IF;

END_FOR
END_GET
END_PROPERTY

{attribute 'monitoring' := 'call'}
PROPERTY Position : LREAL
GET
Position := internalPosition;
END_GET
SET
internalPosition := Position;
END_SET
END_PROPERTY

PROPERTY TrackId : DINT
GET
TrackId := internalTrackId;
END_GET
SET
internalTrackId := TrackId;
END_SET
END_PROPERTY

END_FUNCTION_BLOCK

// ---- POUs/XTS/ErrorMover.TcPOU
{attribute 'hide_all_locals'}
FUNCTION_BLOCK ErrorMover EXTENDS Mover IMPLEMENTS iMover

{attribute 'monitoring' := 'call'}
PROPERTY CurrentDestinationPosition : LREAL
GET


ADSLOGSTR( ADSLOG_MSGTYPE_ERROR, 'The CurrentDestinationPosition Get method has been called on an invalid Mover reference returned by %s.',THIS^.SourceInstancePath);
END_GET
END_PROPERTY

{attribute 'monitoring' := 'call'}
PROPERTY CurrentMoveType : MoverCommandType_enum
GET
VAR
	MoverCurrentMoveType: MoverCommandType_enum;
END_VAR


ADSLOGSTR( ADSLOG_MSGTYPE_ERROR, 'The CurrentMoveType Get method has been called on an invalid Mover reference returned by %s.',THIS^.SourceInstancePath);
END_GET
END_PROPERTY

PROPERTY CurrentObjective : String
GET


ADSLOGSTR( ADSLOG_MSGTYPE_ERROR, 'The CurrentObjective Get method has been called on an invalid Mover reference returned by %s.',THIS^.SourceInstancePath);
END_GET
END_PROPERTY

PROPERTY CurrentTrack : POINTER TO track
GET


ADSLOGSTR( ADSLOG_MSGTYPE_ERROR, 'The CurrentTrack Get method has been called on an invalid Mover reference returned by %s.',THIS^.SourceInstancePath);
END_GET
END_PROPERTY

METHOD Cyclic : iMover
VAR_IN_OUT
	GroupReference		: AXES_GROUP_REF;
END_VAR

VAR
	newCallTime: LREAL;
END_VAR

// If this method was called within the last second, do not write to ADS
newCallTime		:= ULINT_TO_LREAL(F_GetSystemTime())/1E7;

IF ( newCallTime - lastCallCyclic ) > 1 THEN
	ADSLOGSTR( ADSLOG_MSGTYPE_ERROR, 'The Cyclic method has been called on an invalid Mover reference returned by %s.',THIS^.SourceInstancePath);
	lastCallCyclic	:= newCallTime;
END_IF
END_METHOD

METHOD Disable : iMover
VAR_INPUT
END_VAR
VAR
	newCallTime		: LREAL;
END_VAR

// If this method was called within the last second, do not write to ADS
newCallTime		:= ULINT_TO_LREAL(F_GetSystemTime())/1E7;

IF ( newCallTime - lastCallDisable ) > 1 THEN
	ADSLOGSTR( ADSLOG_MSGTYPE_ERROR, 'The Disable method has been called on an invalid Mover reference returned by %s.',THIS^.SourceInstancePath);
	lastCallDisable	:= newCallTime;
END_IF
END_METHOD

METHOD Enable : iMover
VAR_INPUT
END_VAR
VAR
	newCallTime: LREAL;
END_VAR

// If this method was called within the last second, do not write to ADS
newCallTime		:= ULINT_TO_LREAL(F_GetSystemTime())/1E7;

IF ( newCallTime - lastCallEnable ) > 1 THEN
	ADSLOGSTR( ADSLOG_MSGTYPE_ERROR, 'The Enable method has been called on an invalid Mover reference returned by %s.',THIS^.SourceInstancePath);
	lastCallEnable	:= newCallTime;
END_IF
END_METHOD

METHOD GroupStop : iMover
VAR_INPUT
END_VAR
VAR
	newCallTime: LREAL;
END_VAR

// If this method was called within the last second, do not write to ADS
newCallTime		:= ULINT_TO_LREAL(F_GetSystemTime())/1E7;

IF ( newCallTime - lastCallGroupStop ) > 1 THEN
	ADSLOGSTR( ADSLOG_MSGTYPE_ERROR, 'The GroupStop method has been called on an invalid Mover reference returned by %s.',THIS^.SourceInstancePath);
END_IF

lastCallGroupStop	:= newCallTime;
END_METHOD

METHOD Halt : iMover
VAR_INPUT
END_VAR
VAR
	newCallTime: LREAL;
END_VAR

// If this method was called within the last second, do not write to ADS
newCallTime		:= ULINT_TO_LREAL(F_GetSystemTime())/1E7;

IF ( newCallTime - lastCallHalt ) > 1 THEN
	ADSLOGSTR( ADSLOG_MSGTYPE_ERROR, ' The Halt method has been called on an invalid Mover reference returned by %s.',THIS^.SourceInstancePath);
END_IF

lastCallHalt	:= newCallTime;
END_METHOD

{attribute 'monitoring' := 'call'}
PROPERTY IsSyncedToMover : BOOL
GET


ADSLOGSTR( ADSLOG_MSGTYPE_ERROR, 'The IsSyncedToMover Get method has been called on an invalid Mover reference returned by %s.',THIS^.SourceInstancePath);
END_GET
END_PROPERTY

PROPERTY MasterMover : Reference To Mover
GET


ADSLOGSTR( ADSLOG_MSGTYPE_ERROR, 'The MasterMover Get method has been called on an invalid Mover reference returned by %s.',THIS^.SourceInstancePath);
END_GET
END_PROPERTY

METHOD PUBLIC MoveToPosition : iMover
VAR_INPUT
	DestinationPosition		: LREAL;	// position on track for a shuttle to move towards
END_VAR
VAR
	newCallTime				: LREAL;
END_VAR

// If this method was called within the last second, do not write to ADS
newCallTime		:= ULINT_TO_LREAL(F_GetSystemTime())/1E7;

IF ( newCallTime - lastCallMovePos ) > 1 THEN
	ADSLOGSTR( ADSLOG_MSGTYPE_ERROR, 'The MoveToPosition method has been called on an invalid Mover reference returned by %s.',THIS^.SourceInstancePath);
	lastCallMovePos		:= newCallTime;
END_IF
END_METHOD

METHOD MoveToStation : iMover
VAR_INPUT
	DestinationStation	: REFERENCE TO Station;	
END_VAR
VAR
	newCallTime: LREAL;
END_VAR

// If this method was called within the last second, do not write to ADS
newCallTime		:= ULINT_TO_LREAL(F_GetSystemTime())/1E7;

IF ( newCallTime - lastCallMovePos ) > 1 THEN
	ADSLOGSTR( ADSLOG_MSGTYPE_ERROR, 'The MoveToStation method has been called on an invalid Mover reference returned by %s.',THIS^.SourceInstancePath);
	lastCallMovePos		:= newCallTime;
END_IF
END_METHOD

METHOD MoveVelocity : iMover
VAR_INPUT
	DesiredVelocity : LREAL;		//The velocity to be commanded [mm/s]
END_VAR

VAR
	negativeCommand: BOOL;
	newCallTime: LREAL;
END_VAR

// If this method was called within the last second, do not write to ADS
newCallTime		:= ULINT_TO_LREAL(F_GetSystemTime())/1E7;

IF ( newCallTime - lastCallMoveVel ) > 1 THEN
	ADSLOGSTR( ADSLOG_MSGTYPE_ERROR, 'The MoveVelocity method has been called on an invalid Mover reference returned by %s.',THIS^.SourceInstancePath);
	lastCallMoveVel		:= newCallTime;
END_IF
END_METHOD

PROPERTY Payload : Payload_TYP
GET


ADSLOGSTR( ADSLOG_MSGTYPE_ERROR, 'The Payload Get method has been called on an invalid Mover reference returned by %s.',THIS^.SourceInstancePath);
END_GET
SET


ADSLOGSTR( ADSLOG_MSGTYPE_ERROR, 'The Payload Set method has been called on an invalid Mover reference returned by %s.',THIS^.SourceInstancePath);
END_SET
END_PROPERTY

METHOD ReissueCommand : iMover
VAR_INPUT
END_VAR

VAR
	newCallTime: LREAL;
END_VAR

// If this method was called within the last second, do not write to ADS
newCallTime		:= ULINT_TO_LREAL(F_GetSystemTime())/1E7;

IF ( newCallTime - lastCallReissue ) > 1 THEN
	ADSLOGSTR( ADSLOG_MSGTYPE_ERROR, 'The ReissueCommand method has been called on an invalid Mover reference returned by %s.',THIS^.SourceInstancePath);
	lastCallReissue		:= newCallTime;
END_IF
END_METHOD

METHOD SetAcceleration : iMover
VAR_INPUT
	Acceleration	: LREAL;
END_VAR

VAR
	newCallTime: LREAL;
END_VAR

// If this method was called within the last second, do not write to ADS
newCallTime		:= ULINT_TO_LREAL(F_GetSystemTime())/1E7;

IF ( newCallTime - lastCallSetAcc ) > 1 THEN
	ADSLOGSTR( ADSLOG_MSGTYPE_ERROR, 'The SetAcceleration method has been called on an invalid Mover reference returned by %s.',THIS^.SourceInstancePath);
	lastCallSetAcc		:= newCallTime;
END_IF
END_METHOD

METHOD SetDeceleration : iMover
VAR_INPUT
	Deceleration	: LREAL;
END_VAR

VAR
	newCallTime: LREAL;
END_VAR

// If this method was called within the last second, do not write to ADS
newCallTime		:= ULINT_TO_LREAL(F_GetSystemTime())/1E7;

IF ( newCallTime - lastCallSetDec ) > 1 THEN
	ADSLOGSTR( ADSLOG_MSGTYPE_ERROR, 'The SetDeceleration method has been called on an invalid Mover reference returned by %s.',THIS^.SourceInstancePath);
	lastCallSetDec		:= newCallTime;
END_IF
END_METHOD

METHOD SetDirection : iMover
VAR_INPUT
	Direction		: Tc3_Mc3Definitions.MC_Direction;
END_VAR

VAR
	newCallTime: LREAL;
END_VAR

// If this method was called within the last second, do not write to ADS
newCallTime		:= ULINT_TO_LREAL(F_GetSystemTime())/1E7;

IF ( newCallTime - lastCallSetDir ) > 1 THEN
	ADSLOGSTR( ADSLOG_MSGTYPE_ERROR, 'The SetDirection method has been called on an invalid Mover reference returned by %s.',THIS^.SourceInstancePath);
	lastCallSetDir		:= newCallTime;
END_IF
END_METHOD

METHOD SetJerk : iMover
VAR_INPUT
	Jerk		: LREAL;
END_VAR

VAR
	newCallTime: LREAL;
END_VAR

// If this method was called within the last second, do not write to ADS
newCallTime		:= ULINT_TO_LREAL(F_GetSystemTime())/1E7;

IF ( newCallTime - lastCallSetJerk ) > 1 THEN
	ADSLOGSTR( ADSLOG_MSGTYPE_ERROR, 'The SetJerk method has been called on an invalid Mover reference returned by %s.',THIS^.SourceInstancePath);
	lastCallSetJerk		:= newCallTime;
END_IF
END_METHOD

METHOD SetVelocity : iMover
VAR_INPUT
	Velocity	: LREAL;
END_VAR

VAR
	newCallTime: LREAL;
END_VAR

// If this method was called in the last second, do not write to ADS
newCallTime		:= ULINT_TO_LREAL(F_GetSystemTime())/1E7;

IF ( newCallTime - lastCallSetVel ) > 1 THEN
	ADSLOGSTR( ADSLOG_MSGTYPE_ERROR, 'The SetVelocity method has been called on an invalid Mover reference returned by %s.',THIS^.SourceInstancePath);
	lastCallSetVel		:= newCallTime;
END_IF
END_METHOD

METHOD SyncToAxis : iMover
VAR_INPUT
	
	MasterAxis		: REFERENCE TO AXIS_REF;
	MasterSyncPos	: LREAL;	// Master sync position (nonmodulo), where the input axis will be located when first synchronized
	SlaveSyncPos	: LREAL;	// Mover sync position, where the mover will be located when first synchronized
	SyncStrategy	: MC_SYNC_STRATEGY;	// Direction input
	
END_VAR
VAR
	newCallTime		: LREAL;
END_VAR


// If this method was called within the last second, do not write to ADS
newCallTime		:= ULINT_TO_LREAL(F_GetSystemTime())/1E7;

IF (newCallTime - lastCallSync) > 1 THEN
	ADSLOGSTR( ADSLOG_MSGTYPE_ERROR,'The SyncToAxis method has been called on an invalid Mover reference returned by %s',THIS^.SourceInstancePath);
	lastCallSync		:= newCallTime;
END_IF
END_METHOD

METHOD SyncToMover : iMover
VAR_INPUT

	MasterMover		: REFERENCE TO Mover;	// Synchronization master mover, whose position to follow. Further motion commands break the pairing
	Gap				: LREAL;				// Gap distance to lead mover. Positive values indicate following, negative values indicate leading

END_VAR

VAR
	newCallTime: LREAL;
END_VAR

// IF this method was called within the last second, do not write to ADS
newCallTime		:= ULINT_TO_LREAL(F_GetSystemTime())/1E7;

IF ( newCallTime - lastCallSync ) > 1 THEN
	ADSLOGSTR( ADSLOG_MSGTYPE_ERROR, 'The SyncToMover method has been called on an invalid Mover reference returned by %s.',THIS^.SourceInstancePath);
	lastCallSync	:= newCallTime;
END_IF
END_METHOD

END_FUNCTION_BLOCK

// ---- POUs/StarburstDispenser.TcPOU
FUNCTION_BLOCK StarburstDispenser
VAR_INPUT
	mover : Mover;
	timer : TON;
	station_num : INT;
	dispense : BOOL;
	Axis : FB_BasicAxis;
END_VAR
VAR_OUTPUT
	completed : BOOL;
END_VAR
VAR
	aAmount: ARRAY[1..3] OF INT;
	i: INT;
	temp : Payload_TYP;
	seconds: TIME;
	inposition : BOOL := Axis.InPosition;
	count : INT := 0;
	pos : LREAL := Axis.ActualPosition;
	movedistance: LREAL;
	veloc : LREAL := 6000.0;
	state: INT := 0;
END_VAR



completed := FALSE;

//take ou for
// add case




IF dispense THEN
	temp := mover.Payload;
	aAmount[1] := temp.Red;
	aAmount[2] := temp.Orange;
	aAmount[3] := temp.Pink;
	movedistance := (360) * aAmount[station_num];
	
	CASE station_num OF
		
		1: 
			
			Axis.Velocity := 600;
			Axis.MoveRelative(360, TRUE);

		2:
			//motor 2 logic
			timer(IN := TRUE, PT := seconds);
			
		3:
			//motor 3 logic
			timer(IN := TRUE, PT := seconds);
			
		4:
				completed := TRUE;
				Axis.Stop();
		
	END_CASE
END_IF

completed := Timer.Q;
//completed := Axis.InPosition;

IF NOT dispense THEN
	TIMER(IN := FALSE);
	Axis.Stop();
END_IF

END_FUNCTION_BLOCK

// ---- POUs/Orders.TcPOU
PROGRAM Orders
VAR_INPUT
	start: BOOL := FALSE;
END_VAR

VAR
	queue 			: ARRAY[0..9] OF Order_TYP;
	next_empty 		: INT := 0;
	head 			: INT := 0;
	first_order 	: INT := 0;
	size 			: INT := 0;
	MAX_SIZE 		: INT := 10;
	has_order 		: BOOL := FALSE;

	order1 			: Order_TYP;
	order2 			: Order_TYP;
	order3 			: Order_TYP;
	
	
END_VAR

METHOD DEQUEUE : Order_TYP


VAR
	order : Order_TYP;
END_VAR

IF size > 0 THEN
	size := size - 1;
	head := (head + 1) MOD MAX_SIZE;
	
END_IF
END_METHOD

METHOD ENQUEUE : BOOL

VAR_INPUT
    order : Order_TYP; // The order to add
END_VAR
VAR
END_VAR



IF size < MAX_SIZE THEN
	queue[next_empty] := order;
    next_empty := (next_empty + 1) MOD MAX_SIZE; // Increment and wrap around
    size := size + 1;
END_IF
END_METHOD

PROPERTY HasOrder : BOOL
GET
IF size > 0 THEN
	HasOrder := TRUE;
ELSE
	HasOrder := FALSE;
END_IF
END_GET
END_PROPERTY

PROPERTY order : Order_TYP
GET
IF size > 0 THEN
	order := queue[head];
END_IF
END_GET
END_PROPERTY

END_PROGRAM

// ---- VISUs/Controls.TcVIS
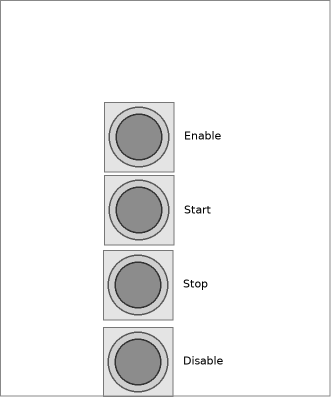
VISUALIZATION Controls  // 331x397
    PushSwitchLed (104,102 70x70), variable: MAIN.MainCommands.Enable, behaviour: TOGGLE, style: Switch-PushSwitchLed-Gray
    Label (181,121 150x30), "Enable"
    Label (181,195 150x30), "Start"
    PushSwitchLed (104,175 70x70), variable: MAIN.MainCommands.Start, behaviour: TOGGLE, style: Switch-PushSwitchLed-Gray
    Label (180,269 150x30), "Stop"
    PushSwitchLed (103,250 70x70), variable: MAIN.MainCommands.Stop, behaviour: TOGGLE, style: Switch-PushSwitchLed-Gray
    Label (180,346 150x30), "Disable"
    PushSwitchLed (103,327 70x70), variable: MAIN.MainCommands.Disable, behaviour: TOGGLE, style: Switch-PushSwitchLed-Gray
END_VISUALIZATION
